FUNCTION_BLOCK LiftSensor (* Template for a simple Basic Function Block Type *)
  (* Standard: 61499-2 *)
  (* Version 1.0, 2019-05-09, jetbrains *)
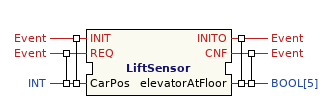
  EVENT_INPUT
    INIT WITH CarPos;
    REQ WITH CarPos; (* Normal Execution Request *)
  END_EVENT
  EVENT_OUTPUT
    INITO WITH elevatorAtFloor;
    CNF WITH elevatorAtFloor; (* Execution Confirmation *)
  END_EVENT
  VAR_INPUT
    CarPos : INT; (* Input event qualifier *)
  END_VAR
  VAR_OUTPUT
    elevatorAtFloor : ARRAY [0..4] OF BOOL;
  END_VAR
  VAR
    prevPos : INT := -1; (* Internal Variable *)
  END_VAR
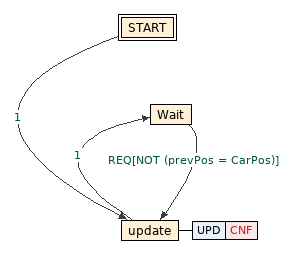
  EC_STATES
    START; (* Initial State *)
    update : UPD -> CNF;
    Wait;
  END_STATES
  EC_TRANSITIONS
    Wait TO update := REQ[NOT (prevPos = CarPos)];
    update TO Wait := 1;
    START TO update := 1;
  END_TRANSITIONS
  ALGORITHM initialize IN ST: (* Initialization algorithm *)
position := CarPos;
  END_ALGORITHM
  ALGORITHM UPD IN ST: (* new algorithm *)
elevatorAtFloor[0] := CarPos = 1;
elevatorAtFloor[1] := CarPos = 3;
elevatorAtFloor[2] := CarPos = 5;
elevatorAtFloor[3] := CarPos = 7;
elevatorAtFloor[4] := CarPos = 9;
prevPos := CarPos;
  END_ALGORITHM
END_FUNCTION_BLOCK
